Staubli VAL3: getTool.pgx

public program getTool(string& x_sTool, tool& x_tTool)
begin
  x_sTool=sToolName
  x_tTool.trsf=tTool[sToolName].trsf
end
